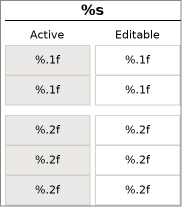
VISUALIZATION VISU_CoverPanelConfig  // 182x207
VAR_IN_OUT
	activeConfig : CoverPanelConfig;
	editableConfig : CoverPanelConfig;
END_VAR
    Textfield (5,75 85x30), "%.1f", text variable: activeConfig.closedPosition, input disabled if: TRUE
        OnMouseClick: write the text variable via Default
    Textfield (5,45 85x30), "%.1f", text variable: activeConfig.openPosition, input disabled if: TRUE
        OnMouseClick: write the text variable via Default
    Textfield (95,75 85x30), "%.1f", text variable: editableConfig.closedPosition, colour toggle: editableConfig.closedPosition <> activeConfig.closedPosition
        OnMouseClick: write the text variable via Default
    Textfield (95,45 85x30), "%.1f", text variable: editableConfig.openPosition, colour toggle: editableConfig.openPosition <> activeConfig.openPosition
        OnMouseClick: write the text variable via Default
    Label (5,25 85x20), "Active"
    Label (95,25 85x20), "Editable"
    Rectangle (5,0 175x20), "%s", text variable: activeConfig.name
    Line (5,20) (180,20)
    Textfield (95,175 85x30), "%.2f", text variable: editableConfig.standstillTolerance, colour toggle: editableConfig.standstillTolerance <> activeConfig.standstillTolerance
        OnMouseClick: write the text variable via Default
    Textfield (5,175 85x30), "%.2f", text variable: activeConfig.standstillTolerance, input disabled if: TRUE
        OnMouseClick: write the text variable via Default
    Textfield (95,145 85x30), "%.2f", text variable: editableConfig.closedTolerance, colour toggle: editableConfig.closedTolerance <> activeConfig.closedTolerance
        OnMouseClick: write the text variable via Default
    Textfield (5,145 85x30), "%.2f", text variable: activeConfig.closedTolerance, input disabled if: TRUE
        OnMouseClick: write the text variable via Default
    Textfield (95,115 85x30), "%.2f", text variable: editableConfig.openTolerance, colour toggle: editableConfig.openTolerance <> activeConfig.openTolerance
        OnMouseClick: write the text variable via Default
    Textfield (5,115 85x30), "%.2f", text variable: activeConfig.openTolerance, input disabled if: TRUE
        OnMouseClick: write the text variable via Default
END_VISUALIZATION

(* stored: Version 1.1.0.1, ProductVersion 3.1.4019.2
   Visu VISU_CoverPanelConfig: Id {743d6c58-5283-4557-a54c-6ca7238f66e2} *)
